// Mitsubishi GX Works2 project: sim   PLC: FX1N/FX1NC

PROGRAM MAIN
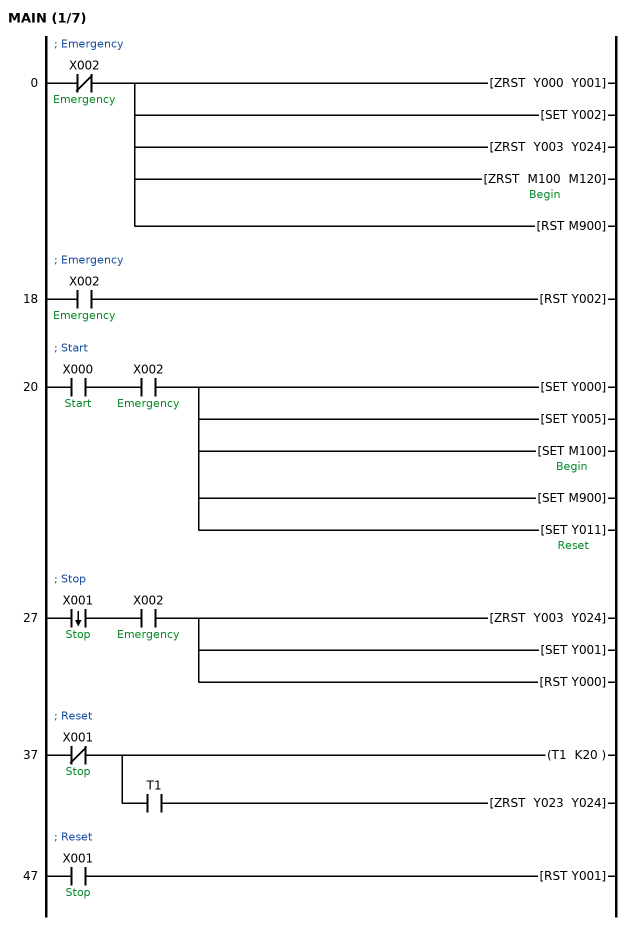
; Emergency
0     LDI     X002  ; Emergency
      ZRST    Y000 Y001
      SET     Y002
      ZRST    Y003 Y024
      ZRST    M100 M120  ; Begin
      RST     M900
; Emergency
18    LD      X002  ; Emergency
      RST     Y002
; Start
20    LD      X000  ; Start
      AND     X002  ; Emergency
      SET     Y000
      SET     Y005
      SET     M100  ; Begin
      SET     M900
      SET     Y011  ; Reset
; Stop
27    LDF     X001  ; Stop
      AND     X002  ; Emergency
      ZRST    Y003 Y024
      SET     Y001
      RST     Y000
; Reset
37    LDI     X001  ; Stop
      OUT     T1 K20
      AND     T1
      ZRST    Y023 Y024
; Reset
47    LD      X001  ; Stop
      RST     Y001
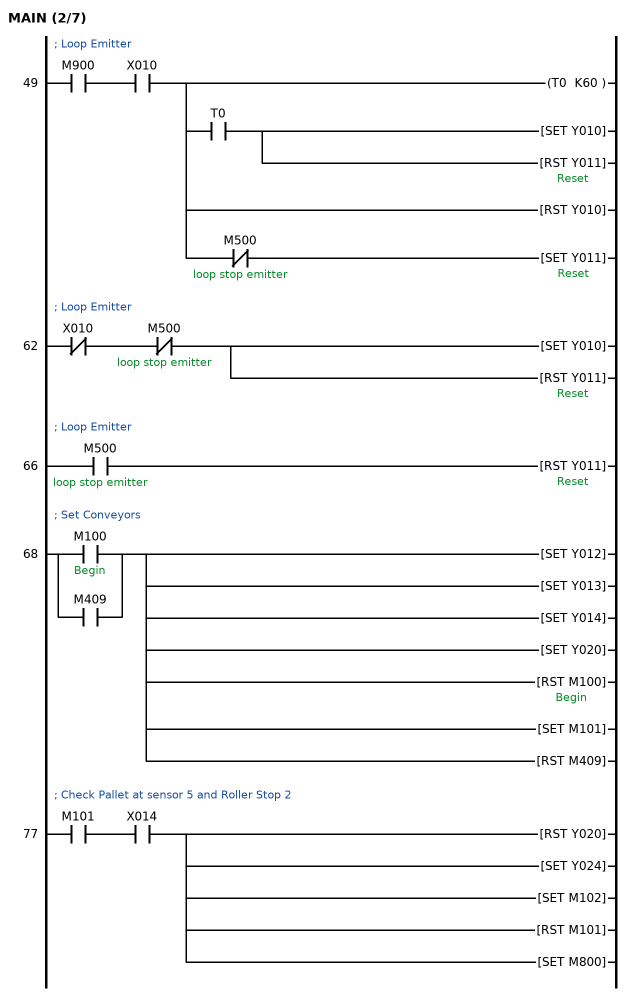
; Loop Emitter
49    LD      M900
      AND     X010
      OUT     T0 K60
      MPS
      AND     T0
      SET     Y010
      RST     Y011  ; Reset
      MPP
      RST     Y010
      ANI     M500  ; loop stop emitter
      SET     Y011  ; Reset
; Loop Emitter
62    LDI     X010
      ANI     M500  ; loop stop emitter
      SET     Y010
      RST     Y011  ; Reset
; Loop Emitter
66    LD      M500  ; loop stop emitter
      RST     Y011  ; Reset
; Set Conveyors
68    LD      M100  ; Begin
      OR      M409
      SET     Y012
      SET     Y013
      SET     Y014
      SET     Y020
      RST     M100  ; Begin
      SET     M101
      RST     M409
; Check Pallet at sensor 5 and Roller Stop 2
77    LD      M101
      AND     X014
      RST     Y020
      SET     Y024
      SET     M102
      RST     M101
      SET     M800
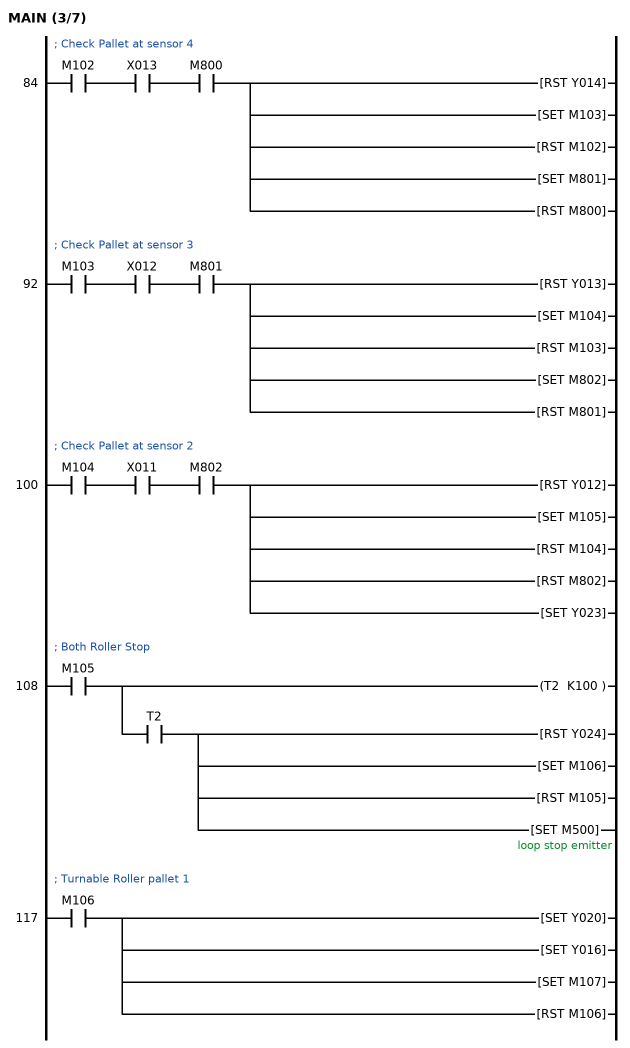
; Check Pallet at sensor 4
84    LD      M102
      AND     X013
      AND     M800
      RST     Y014
      SET     M103
      RST     M102
      SET     M801
      RST     M800
; Check Pallet at sensor 3
92    LD      M103
      AND     X012
      AND     M801
      RST     Y013
      SET     M104
      RST     M103
      SET     M802
      RST     M801
; Check Pallet at sensor 2
100   LD      M104
      AND     X011
      AND     M802
      RST     Y012
      SET     M105
      RST     M104
      RST     M802
      SET     Y023
; Both Roller Stop
108   LD      M105
      OUT     T2 K100
      AND     T2
      RST     Y024
      SET     M106
      RST     M105
      SET     M500  ; loop stop emitter
; Turnable Roller pallet 1
117   LD      M106
      SET     Y020
      SET     Y016
      SET     M107
      RST     M106
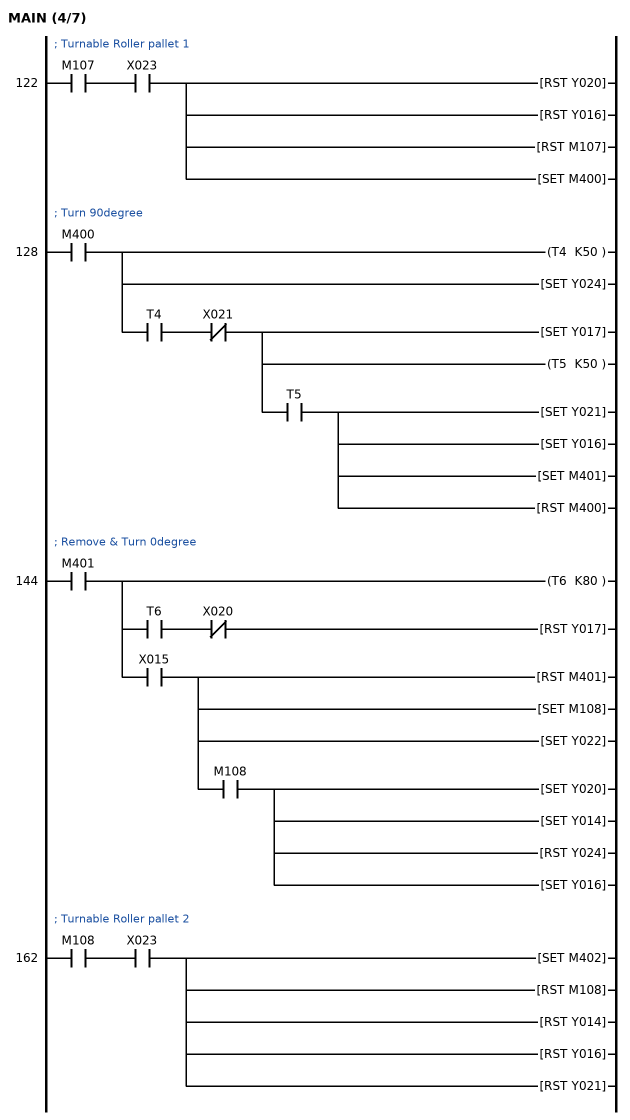
; Turnable Roller pallet 1
122   LD      M107
      AND     X023
      RST     Y020
      RST     Y016
      RST     M107
      SET     M400
; Turn 90degree
128   LD      M400
      OUT     T4 K50
      SET     Y024
      AND     T4
      ANI     X021
      SET     Y017
      OUT     T5 K50
      AND     T5
      SET     Y021
      SET     Y016
      SET     M401
      RST     M400
; Remove & Turn 0degree
144   LD      M401
      OUT     T6 K80
      MPS
      AND     T6
      ANI     X020
      RST     Y017
      MPP
      AND     X015
      RST     M401
      SET     M108
      SET     Y022
      AND     M108
      SET     Y020
      SET     Y014
      RST     Y024
      SET     Y016
; Turnable Roller pallet 2
162   LD      M108
      AND     X023
      SET     M402
      RST     M108
      RST     Y014
      RST     Y016
      RST     Y021
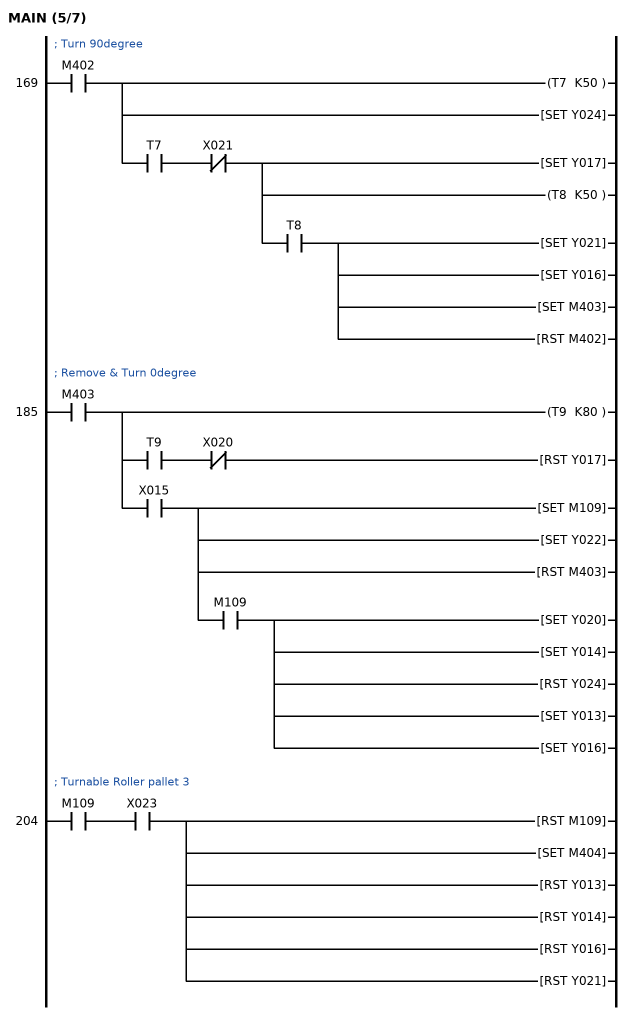
; Turn 90degree
169   LD      M402
      OUT     T7 K50
      SET     Y024
      AND     T7
      ANI     X021
      SET     Y017
      OUT     T8 K50
      AND     T8
      SET     Y021
      SET     Y016
      SET     M403
      RST     M402
; Remove & Turn 0degree
185   LD      M403
      OUT     T9 K80
      MPS
      AND     T9
      ANI     X020
      RST     Y017
      MPP
      AND     X015
      SET     M109
      SET     Y022
      RST     M403
      AND     M109
      SET     Y020
      SET     Y014
      RST     Y024
      SET     Y013
      SET     Y016
; Turnable Roller pallet 3
204   LD      M109
      AND     X023
      RST     M109
      SET     M404
      RST     Y013
      RST     Y014
      RST     Y016
      RST     Y021
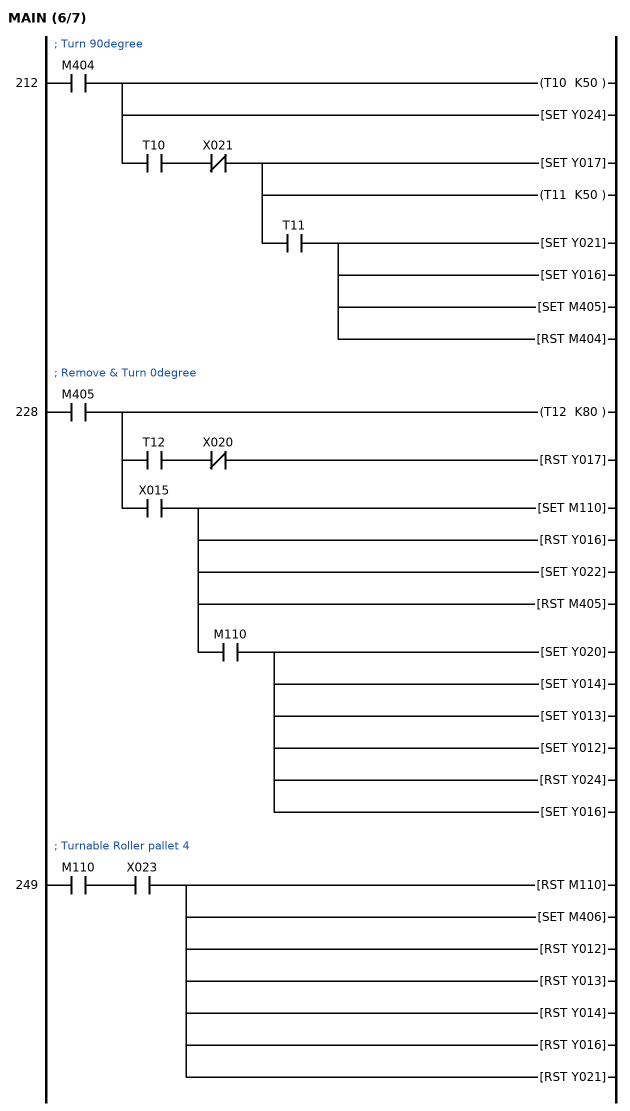
; Turn 90degree
212   LD      M404
      OUT     T10 K50
      SET     Y024
      AND     T10
      ANI     X021
      SET     Y017
      OUT     T11 K50
      AND     T11
      SET     Y021
      SET     Y016
      SET     M405
      RST     M404
; Remove & Turn 0degree
228   LD      M405
      OUT     T12 K80
      MPS
      AND     T12
      ANI     X020
      RST     Y017
      MPP
      AND     X015
      SET     M110
      RST     Y016
      SET     Y022
      RST     M405
      AND     M110
      SET     Y020
      SET     Y014
      SET     Y013
      SET     Y012
      RST     Y024
      SET     Y016
; Turnable Roller pallet 4
249   LD      M110
      AND     X023
      RST     M110
      SET     M406
      RST     Y012
      RST     Y013
      RST     Y014
      RST     Y016
      RST     Y021
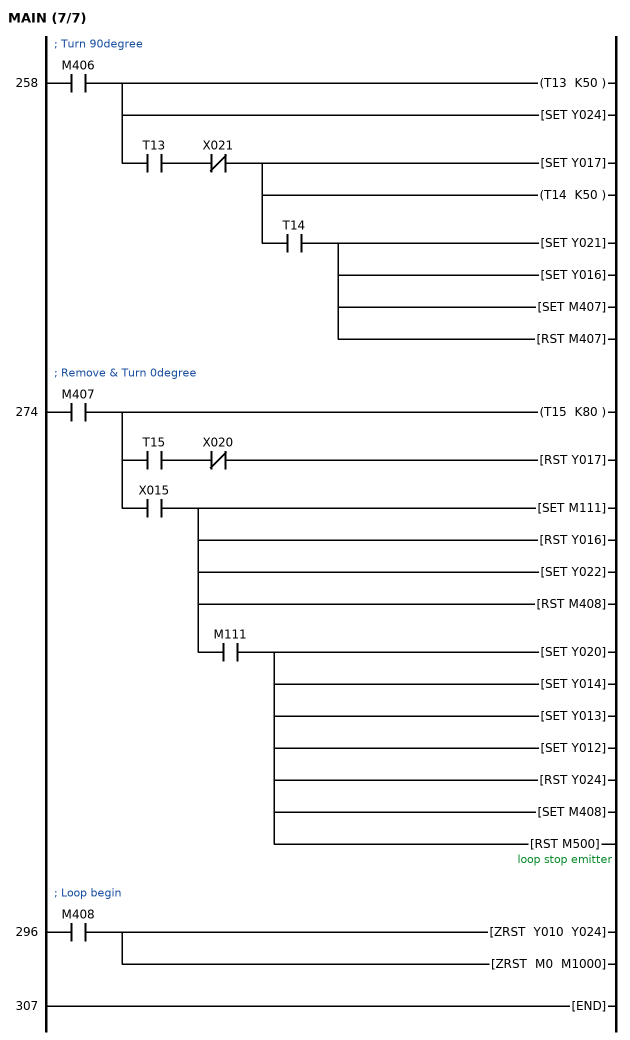
; Turn 90degree
258   LD      M406
      OUT     T13 K50
      SET     Y024
      AND     T13
      ANI     X021
      SET     Y017
      OUT     T14 K50
      AND     T14
      SET     Y021
      SET     Y016
      SET     M407
      RST     M407
; Remove & Turn 0degree
274   LD      M407
      OUT     T15 K80
      MPS
      AND     T15
      ANI     X020
      RST     Y017
      MPP
      AND     X015
      SET     M111
      RST     Y016
      SET     Y022
      RST     M408
      AND     M111
      SET     Y020
      SET     Y014
      SET     Y013
      SET     Y012
      RST     Y024
      SET     M408
      RST     M500  ; loop stop emitter
; Loop begin
296   LD      M408
      ZRST    Y010 Y024
      ZRST    M0 M1000
307   END
END_PROGRAM

// device comments not shown above
X003  ; Emergency
